Staubli VAL3: cognexComm.pjx

--- cognexComm.pjx ---
Parameters version=s7.0 stackSize=5000 millimeterUnit=true
Program file=_incrementCol.pgx
Program file=_toString.pgx
Program file=CheckCellFormat.pgx
Program file=checkColValue.pgx
Program file=coord2Cell.pgx
Program file=getActiveJob.pgx
Program file=getErrorCode.pgx
Program file=getErrorMessage.pgx
Program file=getLibVersion.pgx
Program file=getOnline.pgx
Program file=init.pgx
Program file=loadJob.pgx
Program file=login.pgx
Program file=readErrorTable.pgx
Program file=readLogin.pgx
Program file=readme.pgx
Program file=readNumValue.pgx
Program file=readRect.pgx
Program file=readSocket.pgx
Program file=readStrValue.pgx
Program file=readTrsf.pgx
Program file=saveJob.pgx
Program file=sendCommand.pgx
Program file=setEventAndWait.pgx
Program file=setEventNoWait.pgx
Program file=setOnline.pgx
Program file=start.pgx
Program file=stop.pgx
Program file=trigger.pgx
Program file=writeFloatValue.pgx
Program file=writeIntValue.pgx
Program file=writeSocket.pgx
Program file=writeStrValue.pgx
Data file=cognexComm.dtx

--- READRECT.pgx ---
public program readRect(num nHndl_, string x_sCol, num x_nRow, trsf& trOrigin_[], trsf& trSize_[], bool& x_bResult[])
  local bool l_bIsOK
  local bool l_bResult
begin
  // read X coordinate from spreadsheet
  call readNumValue(nHndl_,x_sCol,x_nRow,trOrigin_.x,x_bResult)
  if x_bResult
    // increment column number
    call _incrementCol(x_sCol,l_bIsOK)
    if l_bIsOK
      // read Y coordinate from spreadsheet
      call readNumValue(nHndl_,x_sCol,x_nRow,trOrigin_.y,x_bResult)
      if x_bResult
        // read width from spreadsheet
        call _incrementCol(x_sCol,l_bIsOK)
        if l_bIsOK
          call readNumValue(nHndl_,x_sCol,x_nRow,trSize_.x,x_bResult)
          if x_bResult
            // read height from spreadsheet
            call _incrementCol(x_sCol,l_bIsOK)
            call readNumValue(nHndl_,x_sCol,x_nRow,trSize_.y,x_bResult)
            if x_bResult
              // read RZ from spreadsheet
              call _incrementCol(x_sCol,l_bIsOK)
              if l_bIsOK
                call readNumValue(nHndl_,x_sCol,x_nRow,trOrigin_.rz,x_bResult)
              endIf
            endIf
          endIf
        endIf
      endIf
    endIf
  endIf
end

--- sendCommand.pgx ---
program sendCommand(num handle_, string cmd_, bool& result_[])
  local string msg
  local bool dummy
  local string str
begin
  // send native command to camera and read command execution result
  call writeSocket(handle_,cmd_)
  call readSocket(handle_,msg,result_)
  str=toNum(msg,errorCode[handle_],dummy)
  result_=errorCode[handle_]==1
  if bDebug
    call getErrorMessage(handle_,msg)
    putln("result: "+msg)
  endIf
end
